{attribute 'linkalways'} 
{attribute 'no_explicit_call' := 'This FB is a CLASS and must be accessed using methods or properties'}
{attribute 'enable_dynamic_creation'}
FUNCTION_BLOCK Node_F_VN_InsertIntoContainer_TcVnKeyPoint EXTENDS VisionNode
VAR
    stElement : _TcVnKeyPoint;
    ipContainer : _ITcVnContainer;
    nIndex : _ULINT(0);
    hrPrev : _HRESULT(S_OK);
    hresult : _HRESULT(S_OK);
END_VAR

METHOD PUBLIC  Clone : I_Node
VAR
	pNode : POINTER TO Node_F_VN_InsertIntoContainer_TcVnKeyPoint;
END_VAR
pNode := __NEW(Node_F_VN_InsertIntoContainer_TcVnKeyPoint);
Clone := pNode^;
END_METHOD

METHOD FB_init : BOOL
VAR_INPUT
	bInitRetains : BOOL; // if TRUE, the retain variables are initialized (warm start / cold start)
	bInCopyCode : BOOL;  // if TRUE, the instance afterwards gets moved into the copy code (online change)
END_VAR
AddInput('stElement', stElement);
AddInput('ipContainer', ipContainer);
AddInput('nIndex', nIndex);
AddInput('hrPrev', hrPrev);
AddOutput('ipContainer', ipContainer);
AddOutput('hresult',hresult);
END_METHOD

METHOD PROTECTED OnExecute : HRESULT
hresult.Value := F_VN_InsertIntoContainer_TcVnKeyPoint(
    stElement := stElement.Value,
    ipContainer := ipContainer.Value,
    nIndex := nIndex.Value,
    hrPrev:= hrPrev.Value);
END_METHOD

METHOD PUBLIC PreExecutionCheck
VAR_INPUT
	Check : I_PreExecutionChecks;
END_VAR
Check.IsTrue(ipContainer.IsValid, 'ipContainer must be a valid container');
END_METHOD

END_FUNCTION_BLOCK

(* stored: Version 1.1.0.1, ProductVersion 3.1.4024.13
   POU Node_F_VN_InsertIntoContainer_TcVnKeyPoint: Id {6f02a3f5-6987-4210-9a3d-6466e42de2fa}, SpecialFunc None
   Folder Constructor: Id {4a26d77c-898c-4d51-a5f0-10dc9fba3973}
   Method Clone: Id {2da56276-03d4-4816-b71a-e5991eaf9cb9}
   Method FB_init: Id {acd022a4-0480-4c30-9de4-b2ab749ad426}
   Method OnExecute: Id {cc379ab1-a82d-47e5-bcfe-b4d79b30cbb9}
   Method PreExecutionCheck: Id {012bc806-e215-457a-9cb3-1c136cf61c2d} *)
